FUNCTION_BLOCK SET_LOCAL_ADS_ADDRESS (* Service Interface Function Block Type *)
  (* Standard: 61499-2; Description: Copyright (c) 2018 TU Vienna/ACIN This program and the accompanying materials are made available under the terms of the Eclipse Public License 2.0 which is available at https://www.eclipse.org/legal/epl-2.0/ SPDX-License-Identifier: EPL-2.0 *)
  (* Version 1.0, 2018-08-31, Martin Melik Merkumians, TU Vienna/ACIN *)
  (* Version 3.0, 2025-04-14, Patrick Aigner, changed package *)
  PACKAGE eclipse4diac::io::ads;
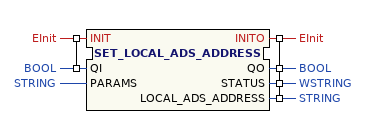
  EVENT_INPUT
    INIT : EInit WITH QI; (* Service Initialization *)
  END_EVENT
  EVENT_OUTPUT
    INITO : EInit WITH QO, STATUS, LOCAL_ADS_ADDRESS; (* Initialization Confirm *)
  END_EVENT
  VAR_INPUT
    QI : BOOL; (* Event Input Qualifier *)
    PARAMS : STRING; (* Local ADS address to set *)
  END_VAR
  VAR_OUTPUT
    QO : BOOL; (* Event Output Qualifier *)
    STATUS : WSTRING; (* Service Status *)
    LOCAL_ADS_ADDRESS : STRING; (* Resulting ADS address *)
  END_VAR
END_FUNCTION_BLOCK
